FUNCTION_BLOCK SubscribeEventHTTP (* Subscribe event using HTTP *)
  (* Standard: 61499-2; Description: Copyright (c) 2019 fortiss GmbH This program and the accompanying materials are made available under the terms of the Eclipse Public License 2.0 which is available at https://www.eclipse.org/legal/epl-2.0/ SPDX-License-Identifier: EPL-2.0 *)
  (* Version 1.0, 2019-09-18, Cabral, fortiss GmbH *)
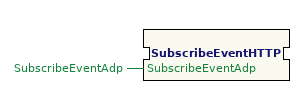
  SOCKETS
    SubscribeEventAdp : SubscribeEventAdp; (* SubscribeEvent adapter *)
  END_SOCKETS
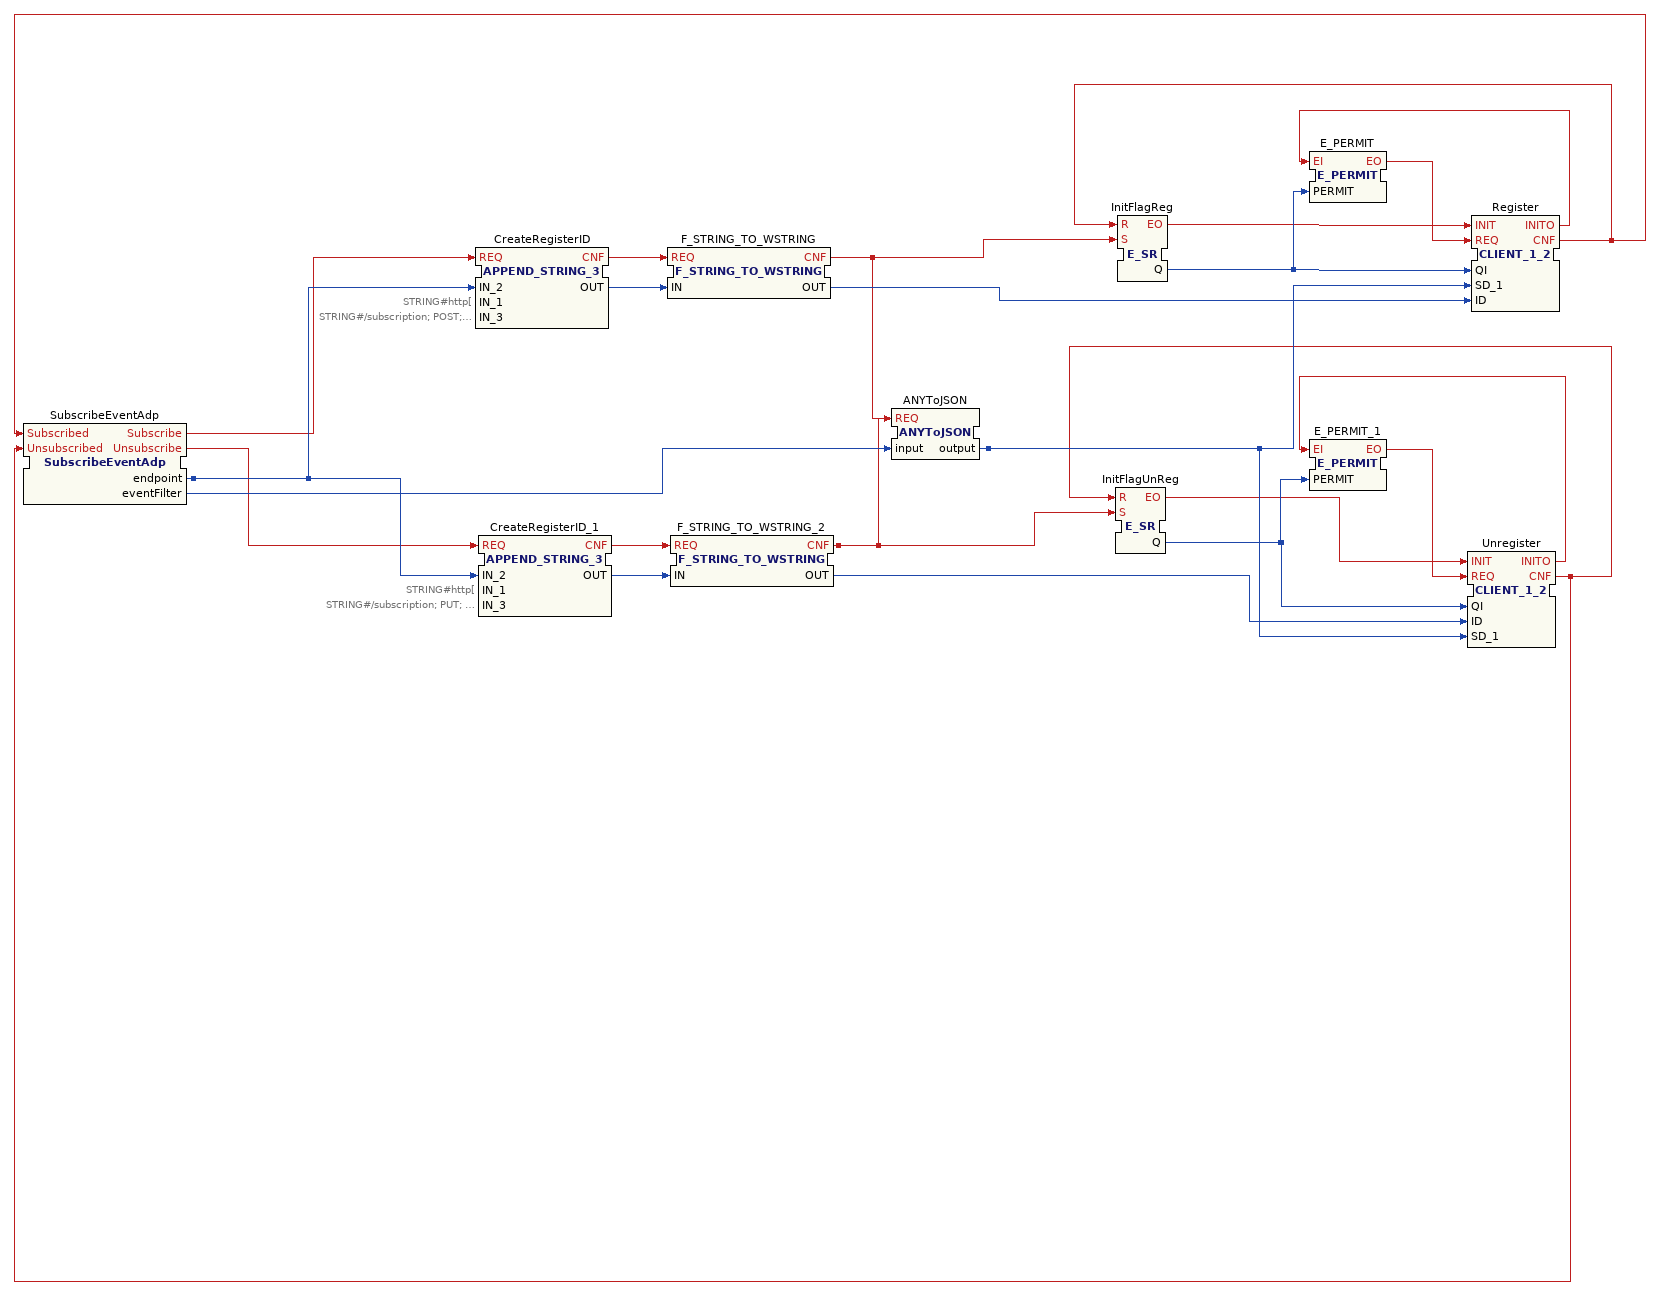
  FBS
    InitFlagReg : E_SR;
    E_PERMIT : E_PERMIT;
    InitFlagUnReg : E_SR;
    F_STRING_TO_WSTRING : F_STRING_TO_WSTRING;
    CreateRegisterID : APPEND_STRING_3(IN_1 := STRING#http[, IN_3 := STRING#/subscription; POST; application/json]);
    ANYToJSON : ANYToJSON;
    E_PERMIT_1 : E_PERMIT;
    Register : CLIENT_1_2;
    Unregister : CLIENT_1_2;
    CreateRegisterID_1 : APPEND_STRING_3(IN_1 := STRING#http[, IN_3 := STRING#/subscription; PUT; application/json]);
    F_STRING_TO_WSTRING_2 : F_STRING_TO_WSTRING;
  END_FBS
  EVENT_CONNECTIONS
    Register.INITO TO E_PERMIT.EI;
    Register.CNF TO InitFlagReg.R;
    InitFlagReg.EO TO Register.INIT;
    CreateRegisterID.CNF TO F_STRING_TO_WSTRING.REQ;
    F_STRING_TO_WSTRING.CNF TO ANYToJSON.REQ;
    E_PERMIT.EO TO Register.REQ;
    F_STRING_TO_WSTRING.CNF TO InitFlagReg.S;
    SubscribeEventAdp.Subscribe TO CreateRegisterID.REQ;
    Register.CNF TO SubscribeEventAdp.Subscribed;
    InitFlagUnReg.EO TO Unregister.INIT;
    E_PERMIT_1.EO TO Unregister.REQ;
    Unregister.INITO TO E_PERMIT_1.EI;
    Unregister.CNF TO SubscribeEventAdp.Unsubscribed;
    Unregister.CNF TO InitFlagUnReg.R;
    SubscribeEventAdp.Unsubscribe TO CreateRegisterID_1.REQ;
    CreateRegisterID_1.CNF TO F_STRING_TO_WSTRING_2.REQ;
    F_STRING_TO_WSTRING_2.CNF TO ANYToJSON.REQ;
    F_STRING_TO_WSTRING_2.CNF TO InitFlagUnReg.S;
  END_CONNECTIONS
  DATA_CONNECTIONS
    InitFlagUnReg.Q TO E_PERMIT_1.PERMIT;
    InitFlagReg.Q TO Register.QI;
    ANYToJSON.output TO Register.SD_1;
    CreateRegisterID.OUT TO F_STRING_TO_WSTRING.IN;
    F_STRING_TO_WSTRING.OUT TO Register.ID;
    InitFlagReg.Q TO E_PERMIT.PERMIT;
    SubscribeEventAdp.endpoint TO CreateRegisterID.IN_2;
    SubscribeEventAdp.eventFilter TO ANYToJSON.input;
    InitFlagUnReg.Q TO Unregister.QI;
    SubscribeEventAdp.endpoint TO CreateRegisterID_1.IN_2;
    CreateRegisterID_1.OUT TO F_STRING_TO_WSTRING_2.IN;
    F_STRING_TO_WSTRING_2.OUT TO Unregister.ID;
    ANYToJSON.output TO Unregister.SD_1;
  END_CONNECTIONS
END_FUNCTION_BLOCK
